FUNCTION_BLOCK DelayDoor (* Template for a simple Basic Function Block Type *)
  (* Standard: 61499-2 *)
  (* Version 1.0, 2019-05-07, jetbrains *)
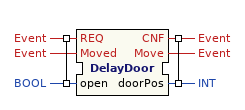
  EVENT_INPUT
    REQ WITH open; (* Normal Execution Request *)
    Moved;
  END_EVENT
  EVENT_OUTPUT
    CNF WITH doorPos; (* Execution Confirmation *)
    Move;
  END_EVENT
  VAR_INPUT
    open : BOOL; (* Input event qualifier *)
  END_VAR
  VAR_OUTPUT
    doorPos : INT; (* Output event qualifier *)
  END_VAR
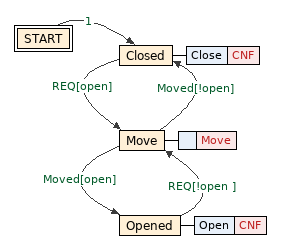
  EC_STATES
    START; (* Initial State *)
    Opened : Open -> CNF;
    Move : -> Move;
    Closed : Close -> CNF;
  END_STATES
  EC_TRANSITIONS
    Opened TO Move := REQ[!open ];
    Move TO Opened := Moved[open];
    START TO Closed := 1;
    Move TO Closed := Moved[!open];
    Closed TO Move := REQ[open];
  END_TRANSITIONS
  ALGORITHM Open IN ST: (* new algorithm *)
doorPos := 10;
  END_ALGORITHM
  ALGORITHM Close IN ST: (* new algorithm *)
doorPos := 0;
  END_ALGORITHM
END_FUNCTION_BLOCK
